// TIA Portal V18 export
TYPE "LaserMarkingBuffer"
// stored: IsFailsafeCompliant false
   STRUCT
      DataMatrixStr : String[60];   // 打标二维码内容
      ProductNameStr : String[60];   // 打标产品名称
      HW_Str : String[60];   // 打标HW内容
      SW_Str : String[60];   // 打标SW内容
      PN_Str : String[60];   // 打标PN内容
      DATA_Str : String[60];   // 打标DATA内容
      SN_Str : String[60];   // 打标SN内容
      ECU_UID_Str : String[60];   // 打标ECU UID内容
      Vdc_Str : String[60];   // 打标电压内容
      Power_Str : String[60];   // 打标功率内容
      Place_Str : String[60];   // 打标产地内容
   END_STRUCT;
END_TYPE
